// TIA Portal V20 export
TYPE "UDT_MTP_ServiceControlExtended"
   STRUCT
      ServiceControl : "UDT_MTP_ServiceControl";
      ServiceSetup { S7_SetPoint := 'True'} : "UDT_Service_Setup";
   END_STRUCT;
END_TYPE
